// TIA Portal V20 export
DATA_BLOCK "JB_Temp"   // DB358
// stored: Access Published, MemoryReserve 100
   VAR
      Test_bypass_Bit : Bool;
      Step_by_Step : Bool;
      Local_Start : Bool;
      Local_Exectue : Bool;
      Local_production : Bool;
      Local_Maintenance : Bool;
      Local_Manual : Bool;
      Local_ClearReset : Bool;
      Local_Stop : Bool;
      Local_mode : Bool;
      resultOK : Bool;
      resultNG : Bool;
      Simulation_initializing : Bool;
      Simulation_On : Bool;
      Test_Homing : Array[0..20] of Bool;
      Test_sig_0 : Array[1..9] of Bool;
      Test_sig_1 : Array[1..9] of Bool;
      Test_sig_2 : Array[1..2, 0..10, 0..10] of Bool;
      Test_sig_3 : Array[1..3, 0..10, 0..10] of Bool;
      Test_sig_4 : Array[1..3, 0..10, 0..10] of Bool;
      Test_sig_5 : Array[1..3, 0..10, 0..10] of Bool;
      Test_sig_6 : Array[1..9, 0..10] of Bool;
      Test_sig_7 : Array[1..9, 0..10] of Bool;
      Test_sig_8 : Array[1..4, 0..10] of Bool;
      Test_sig_9 : Array[1..2, 0..10] of Bool;
      Test_sig_10 : Array[1..9] of Bool;
      Test_sig_11 : Array[1..9] of Bool;
      Test_sig_12 : Array[1..9] of Bool;
      Test_sig_13 : Array[1..9, 0..10] of Bool;
      Suspend : Bool;
      Abort : Bool;
      Hold : Bool;
   END_VAR
BEGIN
END_DATA_BLOCK
